PROGRAM originRepo
VAR
END_VAR

END_PROGRAM

(* stored: Version 1.1.0.1, ProductVersion 3.1.4024.12
   POU originRepo: Id {b4668f6f-2cb5-0ea5-249d-7446f2c7583a}, SpecialFunc None *)
